FUNCTION_BLOCK FB_MaterialDensityLookup_Test EXTENDS TcUnit.FB_TestSuite
VAR
END_VAR


GivenElementExpectCorrectDensity();


METHOD PRIVATE GivenElementExpectCorrectDensity
VAR
    fResult : LREAL;
END_VAR

TEST('GivenElementExpectCorrectDensity');

fResult := F_MaterialDensityLookup(
    sMaterialName := 'C (Diamond)'
);

AssertEquals_LREAL(
    Expected := 3.51,
    Actual := fResult,
    Delta := 1e-9,
    Message := 'Incorrect result.'
);

TEST_FINISHED();
END_METHOD

END_FUNCTION_BLOCK

(* stored: Version 1.1.0.1
   POU FB_MaterialDensityLookup_Test: Id {e51ca4d4-f0f4-4934-bf8a-ed7cf37c61a4}, SpecialFunc None
   Method GivenElementExpectCorrectDensity: Id {1e8c377a-f780-42e4-9353-5fff4c69f82e} *)
